FUNCTION_BLOCK FB_Publisher IMPLEMENTS I_EventPublisher
VAR
	raiseEvent						: BOOL;
	_event							: INT;
	_eventPrev						: INT;
	
	publisher						: FB_Observable;	
END_VAR

IF _eventPrev <> _event 			THEN
	publisher.notify();
	_eventPrev := _event;
END_IF

METHOD attach : BOOL
VAR_INPUT
	observer			: I_Observer;
END_VAR
attach := publisher.attach(observer);
END_METHOD

METHOD detach : BOOL
VAR_INPUT
	observer	: I_Observer;
END_VAR
detach := publisher.detach(observer);
END_METHOD

PROPERTY event : int
GET
event := _event;
END_GET
END_PROPERTY

END_FUNCTION_BLOCK

(* stored: Version 1.1.0.1, ProductVersion 3.1.4024.11
   POU FB_Publisher: Id {270e0f21-f10c-4d6e-aaab-748f1b75e82c}, SpecialFunc None
   Method attach: Id {ab4ff1ed-f2e9-459d-bd43-c6901c9fa429}
   Method detach: Id {0aef42ef-b37c-48ca-9ad5-1143c99045a0}
   Property event: Id {5a53bf6d-f733-4ff7-bc62-c7e9a7ce7ec4}
   Get Get: Id {cdadf8c7-7fab-4fb4-84ee-b1e660efac40} *)
